{attribute 'no-analysis'}
TYPE ST_EL3443_DPM_VariantValues :
STRUCT
	astLx 			: ARRAY[1..3] OF ST_EL3443_DPM_VariantLx;
	stTotal 		: ST_EL3443_DPM_VariantTotal;
END_STRUCT
END_TYPE

(* stored: Version 1.1.0.1, ProductVersion 3.1.4024.4
   DUT ST_EL3443_DPM_VariantValues: Id {813e8971-4aed-4e9c-b1a0-00d3673f0cca} *)
